(* LEFT function for long string *)
FUNCTION F_LongLEFT : T_LongSTRING
VAR_INPUT
	strString			: T_LongSTRING;
	nLen				: UINT;	(* no of chars to extract *)
END_VAR
VAR
	nStringLen			: UINT;
	nActLen				: UINT;
END_VAR
(*
-------------------------------------------------------------------------------------------------
DATE		Version	Author	Comments
-------------------------------------------------------------------------------------------------
30/01/2015	3.00.00	PB		Initial release

-------------------------------------------------------------------------------------------------
*)

(* length of input string *)
nStringLen := TO_UINT(LEN2(ADR(strString)));

(* input string length <= 255 chars *)
IF nStringLen <= 255 THEN

	(* use standard LEFT function *)
	F_LongLEFT := LEFT(strString, TO_INT(nLen));

(* input string length > 255 chars *)
ELSE

	(* no of chars specified *)
	IF nLen > 0 AND nStringLen > 0 THEN

		(* chars required < strString length *)
		IF nLen < nStringLen THEN

			(* clamp no of chars to be extracted to length of input string *)
			nActLen := MIN(nLen, nStringLen);
	
			(* extract chars from strString *)
			MEMMOVE(ADR(F_LongLEFT), ADR(strString), nActLen);
	
			(* set last char to 16#00 to terminate the string with NULL *)
			MEMSET(ADR(F_LongLEFT) + nActLen, 16#00, 1);

		(* chars required >= strString length *)
		ELSE

			(* return complete string *)
			F_LongLEFT := strString;
		END_IF

	(* no length specified *)
	ELSE

		(* return empty string *)
		F_LongLEFT := '';
	END_IF
END_IF

END_FUNCTION

(* stored: Version 1.1.0.1
   POU F_LongLEFT: Id {d3ed8215-92ef-45b4-9c10-f236d84d8beb}, SpecialFunc None *)
